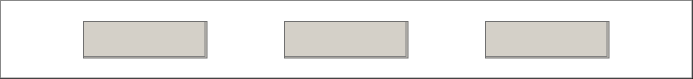
VISUALIZATION VISU_AXE_STD1_FCT_MANU  // 693x79
VAR_IN_OUT
	m_Input_MOTEUR: BLOCK_AXE_STD1;
	m_Input_PRG_MOUVEMENT_PS: BLOCK_PRG_MOUVEMENT_PS;
END_VAR
VAR_INPUT
	m_Input_INDEX_MOTEUR : INT;
END_VAR
    Rectangle (0,0 693x79)
    Button (83,21 124x37), invisible if: NOT .PRG_USER.ACTU_USER.MAINTENANCE OR NOT m_Input_MOTEUR.MANUAL, text list: 'TextList_Moteurs', text index: 0
        tap m_Input_MOTEUR.CO_RESET
    Button (284,21 124x37), invisible if: NOT PRG_USER.ACTU_USER.MAINTENANCE OR NOT m_Input_MOTEUR.MANUAL OR NOT m_Input_MOTEUR.CONF_No_Ref, input disabled if: NOT m_Input_MOTEUR.OP_Validation.AR, text list: 'TextList_Moteurs', text index: 1
        tap m_Input_MOTEUR.M_BIAS
    Button (485,21 124x37), invisible if: NOT PRG_USER.ACTU_USER.MAINTENANCE OR NOT m_Input_MOTEUR.MANUAL OR NOT m_Input_PRG_MOUVEMENT_PS.CONF_Jog[m_Input_INDEX_MOTEUR], text list: 'TextList_Moteurs', text index: 2
        tap m_Input_MOTEUR.CO_Devalid
END_VISUALIZATION

(* stored: Version 1.1.0.1, ProductVersion 3.1.4024.10
   Visu VISU_AXE_STD1_FCT_MANU: Id {0f611c8b-6665-4334-aee4-2e784cd01cbb} *)
